{attribute 'OPC.UA.DA.StructuredType' := '1'}
FUNCTION_BLOCK FB_PumpDOL_Onga413 EXTENDS FB_BaseDevice IMPLEMENTS I_Device, I_PumpVSD

VAR
	{attribute 'OPC.UA.DA' := '1'} 
	bInContactor AT %I*: BOOL := FALSE;
	{attribute 'OPC.UA.DA' := '1'} 
	bOutContactor AT %Q*: BOOL := FALSE;


	//MB:  REFERENCE TO FB_ModbusMaster;
	{attribute 'OPC.UA.DA' := '1'} 
	nFrequencySetPoint: REAL := 0;
	{attribute 'OPC.UA.DA' := '1'} 
	nFrequencyActual: REAL := 0;
	
	{attribute 'OPC.UA.DA' := '0'} 
	eSMState: (WAIT, STARTING, RUNNING, STOPPING, STOPPED);
	
END_VAR

fbTONstartTime();
fbTONstopTime();

IF GVL.bAutoUpdateDeviceState THEN
	eState := eStateTarget;	
END_IF



IF bEnable THEN
	IF eStateTarget = E_DeviceState.ON AND eState <> E_DeviceState.ON THEN
		eSMState := STARTING;
	END_IF
END_IF

IF eStateTarget = E_DeviceState.OFF AND eState <> E_DeviceState.OFF THEN
		eSMState := STOPPING;
END_IF


CASE eSMState OF
	
	WAIT:
		//Wait for method call to change ESMState
		
	STARTING: 
		eState := E_DeviceState.STARTING;

		bOutContactor := TRUE;
	
		IF fbTONstartTime.Q THEN
			eSMState := WAIT;
			raiseAlarm(Priority := E_AlarmPriority.High, Label := 'Failed to Start', Enabled := TRUE, DeviceAlarmID := 2);
		END_IF
		
		IF bInContactor THEN
			eSMState := RUNNING;
			eState := E_DeviceState.RUNNING;
		END_IF
		
	RUNNING:
		IF bInContactor <> TRUE THEN
			raiseAlarm(Priority := E_AlarmPriority.High, Label := 'Power Lost', Enabled := TRUE, DeviceAlarmID := 2);
			eState := E_DeviceState.FAULTED;
			eSMState := WAIT;
		END_IF
		
		// Add pump / motor control here - look at built in Twincat libraries 
		// Add relevant VSD signals to check
		

	STOPPING:
		eState := E_DeviceState.STOPPING;
		bOutContactor := FALSE;
				
		IF fbTONstopTime.Q THEN
			eSMState := WAIT;
			raiseAlarm(Priority := E_AlarmPriority.High, Label := 'Failed to Stop', Enabled := TRUE, DeviceAlarmID := 3);
		END_IF 
		
		IF bInContactor = FALSE AND nFrequencyActual = 0 THEN
			eSMState := STOPPED;	
		END_IF
		

	STOPPED:
		eState := E_DeviceState.IDLE;
		eSMState := WAIT;
		
		
END_CASE

{warning 'add method implementation '}
METHOD disable : BOOL
END_METHOD

{warning 'add method implementation '}
METHOD enable : BOOL
END_METHOD

{warning 'add method implementation '}
METHOD FB_init : BOOL
VAR_INPUT
	(* if TRUE, the retain variables are initialized (warm start / cold start)*)
	bInitRetains	: BOOL;
	(* if TRUE, the instance afterwards gets moved into the copy code (online change)*)
	bInCopyCode	: BOOL;
	PumpID	: STRING(80);
	PumpDescr	: STRING(255);
END_VAR
sID := PumpID;
sDescr := PumpDescr;
END_METHOD

{warning 'add method implementation '}
METHOD getFrequency : REAL
END_METHOD

METHOD setModbusMaster : BOOL
METHOD setModbusMaster : BOOL
VAR_INPUT
	//ModbusMaster: REFERENCE TO FB_ModbusMaster;
END_VAR
//MB := ModbusMaster;
END_METHOD

METHOD setOff : BOOL
VAR_INPUT
END_VAR
END_METHOD

METHOD setOn : BOOL
VAR_INPUT
END_VAR
END_METHOD

{warning 'add method implementation '}
METHOD setReference : BOOL
VAR_INPUT
	RefSetPoint	: REAL;
END_VAR
END_METHOD

END_FUNCTION_BLOCK

(* stored: Version 1.1.0.1, ProductVersion 3.1.4024.12
   POU FB_PumpDOL_Onga413: Id {98d36f57-66f2-43c3-a9f8-333f76688db4}, SpecialFunc None
   Method disable: Id {52184ce4-ba51-492f-8b16-9d6aa7f869d7}
   Method enable: Id {e71dcaf9-338a-4ee2-8469-1ce0297f1667}
   Method FB_init: Id {a509d217-6b91-4892-9851-1386595f7c5a}
   Method getFrequency: Id {1bd0517e-c9f7-4f28-ba96-b1d1897dbac0}
   Method setModbusMaster: Id {8bb2eba5-78c9-48b5-88ae-9944c4a8a375}
   Method setOff: Id {5c03639b-ce96-4c20-8db4-a9f7040b541e}
   Method setOn: Id {a5183cc9-513b-4b74-aad8-b0c8dddf7764}
   Method setReference: Id {5d727785-f31f-45c7-a65f-6eb9618b8130} *)
